TYPE T_Ctrl_SIf_PLS_Out :
STRUCT
END_STRUCT
END_TYPE

(* stored: Version 1.1.0.1, ProductVersion 3.1.0.19
   DUT T_Ctrl_SIf_PLS_Out: Id {9ea34203-0c76-4c6c-a0b5-a51c508070f4} *)
